{attribute 'qualified_only'}
{attribute 'strict'}
{attribute 'to_string'}
TYPE E_APP_VARIANT :
(
  VARIANT_INVALID,
	VARIANT_OUTPUT_24,
  VARIANT_OUTPUT_CLAMP
);
END_TYPE

(* stored: Version 1.1.0.1, ProductVersion 3.1.4026.13
   DUT E_APP_VARIANT: Id {c60fa34a-3e86-4863-a8f4-13e1223a017e} *)
